// TIA Portal V20 export
DATA_BLOCK "instGetIdentRf"   // DB217
// stored: InstanceOfName GetIdentRf, InstanceOfType FB
"GetIdentRf"
   // VAR_INPUT
   //    identRfAllUnits { ExternalAccessible := 'False'; ExternalVisible := 'False'; ExternalWritable := 'False'} : Array[0.."NO_OF_UNITS"] of "typeEMIdentRf";
   //    numberOfRfReaders : USInt := 1;
   // END_VAR
   // VAR_OUTPUT
   //    selectedUnit : USInt := 1;
   //    selectedEM : USInt := 6;
   //    error : Word := 16#7001;
   // END_VAR
   // VAR_IN_OUT
   //    IdentRfInterfaceHmi : "typeIdentRfHmi";
   // END_VAR
   // VAR
   //    statSelectedEMIdentRf : USInt := 6;
   //    statSelectedUnitIdentRf : USInt := 1;
   // END_VAR
BEGIN
   identRfAllUnits[0].identRfEM[0..7].selectedUnit := 0;
   identRfAllUnits[0].identRfEM[0..7].selectedEM := 0;
   identRfAllUnits[0].identRfEM[0..7].rfReaderId := 0;
   identRfAllUnits[0].identRfEM[0..7].numberOfRf := 0;
   identRfAllUnits[0].identRfEM[0].rfReader[0..1].deviceName := WSTRING#'';
   identRfAllUnits[0].identRfEM[1].rfReader[0..1].deviceName := WSTRING#'';
   identRfAllUnits[0].identRfEM[2].rfReader[0..1].deviceName := WSTRING#'';
   identRfAllUnits[0].identRfEM[3].rfReader[0..1].deviceName := WSTRING#'';
   identRfAllUnits[0].identRfEM[4].rfReader[0..1].deviceName := WSTRING#'';
   identRfAllUnits[0].identRfEM[5].rfReader[0..1].deviceName := WSTRING#'';
   identRfAllUnits[0].identRfEM[6].rfReader[0..1].deviceName := WSTRING#'';
   identRfAllUnits[0].identRfEM[7].rfReader[0..1].deviceName := WSTRING#'';
   identRfAllUnits[0].identRfEM[0].rfReader[0..1].deviceType := WSTRING#'';
   identRfAllUnits[0].identRfEM[1].rfReader[0..1].deviceType := WSTRING#'';
   identRfAllUnits[0].identRfEM[2].rfReader[0..1].deviceType := WSTRING#'';
   identRfAllUnits[0].identRfEM[3].rfReader[0..1].deviceType := WSTRING#'';
   identRfAllUnits[0].identRfEM[4].rfReader[0..1].deviceType := WSTRING#'';
   identRfAllUnits[0].identRfEM[5].rfReader[0..1].deviceType := WSTRING#'';
   identRfAllUnits[0].identRfEM[6].rfReader[0..1].deviceType := WSTRING#'';
   identRfAllUnits[0].identRfEM[7].rfReader[0..1].deviceType := WSTRING#'';
   identRfAllUnits[0].identRfEM[0].rfReader[0..1].deviceId := 0;
   identRfAllUnits[0].identRfEM[1].rfReader[0..1].deviceId := 0;
   identRfAllUnits[0].identRfEM[2].rfReader[0..1].deviceId := 0;
   identRfAllUnits[0].identRfEM[3].rfReader[0..1].deviceId := 0;
   identRfAllUnits[0].identRfEM[4].rfReader[0..1].deviceId := 0;
   identRfAllUnits[0].identRfEM[5].rfReader[0..1].deviceId := 0;
   identRfAllUnits[0].identRfEM[6].rfReader[0..1].deviceId := 0;
   identRfAllUnits[0].identRfEM[7].rfReader[0..1].deviceId := 0;
   identRfAllUnits[0].identRfEM[0].rfReader[0..1].tagType := WSTRING#'';
   identRfAllUnits[0].identRfEM[1].rfReader[0..1].tagType := WSTRING#'';
   identRfAllUnits[0].identRfEM[2].rfReader[0..1].tagType := WSTRING#'';
   identRfAllUnits[0].identRfEM[3].rfReader[0..1].tagType := WSTRING#'';
   identRfAllUnits[0].identRfEM[4].rfReader[0..1].tagType := WSTRING#'';
   identRfAllUnits[0].identRfEM[5].rfReader[0..1].tagType := WSTRING#'';
   identRfAllUnits[0].identRfEM[6].rfReader[0..1].tagType := WSTRING#'';
   identRfAllUnits[0].identRfEM[7].rfReader[0..1].tagType := WSTRING#'';
   identRfAllUnits[0].identRfEM[0].rfReader[0..1].cameraMode := WSTRING#'';
   identRfAllUnits[0].identRfEM[1].rfReader[0..1].cameraMode := WSTRING#'';
   identRfAllUnits[0].identRfEM[2].rfReader[0..1].cameraMode := WSTRING#'';
   identRfAllUnits[0].identRfEM[3].rfReader[0..1].cameraMode := WSTRING#'';
   identRfAllUnits[0].identRfEM[4].rfReader[0..1].cameraMode := WSTRING#'';
   identRfAllUnits[0].identRfEM[5].rfReader[0..1].cameraMode := WSTRING#'';
   identRfAllUnits[0].identRfEM[6].rfReader[0..1].cameraMode := WSTRING#'';
   identRfAllUnits[0].identRfEM[7].rfReader[0..1].cameraMode := WSTRING#'';
   identRfAllUnits[0].identRfEM[0].rfReader[0..1].resultState := WSTRING#'';
   identRfAllUnits[0].identRfEM[1].rfReader[0..1].resultState := WSTRING#'';
   identRfAllUnits[0].identRfEM[2].rfReader[0..1].resultState := WSTRING#'';
   identRfAllUnits[0].identRfEM[3].rfReader[0..1].resultState := WSTRING#'';
   identRfAllUnits[0].identRfEM[4].rfReader[0..1].resultState := WSTRING#'';
   identRfAllUnits[0].identRfEM[5].rfReader[0..1].resultState := WSTRING#'';
   identRfAllUnits[0].identRfEM[6].rfReader[0..1].resultState := WSTRING#'';
   identRfAllUnits[0].identRfEM[7].rfReader[0..1].resultState := WSTRING#'';
   identRfAllUnits[0].identRfEM[0].rfReader[0..1].progNo := 0;
   identRfAllUnits[0].identRfEM[1].rfReader[0..1].progNo := 0;
   identRfAllUnits[0].identRfEM[2].rfReader[0..1].progNo := 0;
   identRfAllUnits[0].identRfEM[3].rfReader[0..1].progNo := 0;
   identRfAllUnits[0].identRfEM[4].rfReader[0..1].progNo := 0;
   identRfAllUnits[0].identRfEM[5].rfReader[0..1].progNo := 0;
   identRfAllUnits[0].identRfEM[6].rfReader[0..1].progNo := 0;
   identRfAllUnits[0].identRfEM[7].rfReader[0..1].progNo := 0;
   identRfAllUnits[0].identRfEM[0].rfReader[0..1].progNumberWrite := 0;
   identRfAllUnits[0].identRfEM[1].rfReader[0..1].progNumberWrite := 0;
   identRfAllUnits[0].identRfEM[2].rfReader[0..1].progNumberWrite := 0;
   identRfAllUnits[0].identRfEM[3].rfReader[0..1].progNumberWrite := 0;
   identRfAllUnits[0].identRfEM[4].rfReader[0..1].progNumberWrite := 0;
   identRfAllUnits[0].identRfEM[5].rfReader[0..1].progNumberWrite := 0;
   identRfAllUnits[0].identRfEM[6].rfReader[0..1].progNumberWrite := 0;
   identRfAllUnits[0].identRfEM[7].rfReader[0..1].progNumberWrite := 0;
   identRfAllUnits[0].identRfEM[0].rfReader[0..1].pushbutton := 16#0000;
   identRfAllUnits[0].identRfEM[1].rfReader[0..1].pushbutton := 16#0000;
   identRfAllUnits[0].identRfEM[2].rfReader[0..1].pushbutton := 16#0000;
   identRfAllUnits[0].identRfEM[3].rfReader[0..1].pushbutton := 16#0000;
   identRfAllUnits[0].identRfEM[4].rfReader[0..1].pushbutton := 16#0000;
   identRfAllUnits[0].identRfEM[5].rfReader[0..1].pushbutton := 16#0000;
   identRfAllUnits[0].identRfEM[6].rfReader[0..1].pushbutton := 16#0000;
   identRfAllUnits[0].identRfEM[7].rfReader[0..1].pushbutton := 16#0000;
   identRfAllUnits[0].identRfEM[0].rfReader[0..1].enablePushbutton := 16#0000;
   identRfAllUnits[0].identRfEM[1].rfReader[0..1].enablePushbutton := 16#0000;
   identRfAllUnits[0].identRfEM[2].rfReader[0..1].enablePushbutton := 16#0000;
   identRfAllUnits[0].identRfEM[3].rfReader[0..1].enablePushbutton := 16#0000;
   identRfAllUnits[0].identRfEM[4].rfReader[0..1].enablePushbutton := 16#0000;
   identRfAllUnits[0].identRfEM[5].rfReader[0..1].enablePushbutton := 16#0000;
   identRfAllUnits[0].identRfEM[6].rfReader[0..1].enablePushbutton := 16#0000;
   identRfAllUnits[0].identRfEM[7].rfReader[0..1].enablePushbutton := 16#0000;
   identRfAllUnits[0].identRfEM[0].rfReader[0..1].status := 16#0000;
   identRfAllUnits[0].identRfEM[1].rfReader[0..1].status := 16#0000;
   identRfAllUnits[0].identRfEM[2].rfReader[0..1].status := 16#0000;
   identRfAllUnits[0].identRfEM[3].rfReader[0..1].status := 16#0000;
   identRfAllUnits[0].identRfEM[4].rfReader[0..1].status := 16#0000;
   identRfAllUnits[0].identRfEM[5].rfReader[0..1].status := 16#0000;
   identRfAllUnits[0].identRfEM[6].rfReader[0..1].status := 16#0000;
   identRfAllUnits[0].identRfEM[7].rfReader[0..1].status := 16#0000;
   identRfAllUnits[0].identRfEM[0].rfReader[0..1].alarmCategorie := 0;
   identRfAllUnits[0].identRfEM[1].rfReader[0..1].alarmCategorie := 0;
   identRfAllUnits[0].identRfEM[2].rfReader[0..1].alarmCategorie := 0;
   identRfAllUnits[0].identRfEM[3].rfReader[0..1].alarmCategorie := 0;
   identRfAllUnits[0].identRfEM[4].rfReader[0..1].alarmCategorie := 0;
   identRfAllUnits[0].identRfEM[5].rfReader[0..1].alarmCategorie := 0;
   identRfAllUnits[0].identRfEM[6].rfReader[0..1].alarmCategorie := 0;
   identRfAllUnits[0].identRfEM[7].rfReader[0..1].alarmCategorie := 0;
   identRfAllUnits[0].identRfEM[0].rfReader[0..1].alarmNo := 0;
   identRfAllUnits[0].identRfEM[1].rfReader[0..1].alarmNo := 0;
   identRfAllUnits[0].identRfEM[2].rfReader[0..1].alarmNo := 0;
   identRfAllUnits[0].identRfEM[3].rfReader[0..1].alarmNo := 0;
   identRfAllUnits[0].identRfEM[4].rfReader[0..1].alarmNo := 0;
   identRfAllUnits[0].identRfEM[5].rfReader[0..1].alarmNo := 0;
   identRfAllUnits[0].identRfEM[6].rfReader[0..1].alarmNo := 0;
   identRfAllUnits[0].identRfEM[7].rfReader[0..1].alarmNo := 0;
   identRfAllUnits[0].identRfEM[0].rfReader[0..1].alarmCode := 16#0000_0000;
   identRfAllUnits[0].identRfEM[1].rfReader[0..1].alarmCode := 16#0000_0000;
   identRfAllUnits[0].identRfEM[2].rfReader[0..1].alarmCode := 16#0000_0000;
   identRfAllUnits[0].identRfEM[3].rfReader[0..1].alarmCode := 16#0000_0000;
   identRfAllUnits[0].identRfEM[4].rfReader[0..1].alarmCode := 16#0000_0000;
   identRfAllUnits[0].identRfEM[5].rfReader[0..1].alarmCode := 16#0000_0000;
   identRfAllUnits[0].identRfEM[6].rfReader[0..1].alarmCode := 16#0000_0000;
   identRfAllUnits[0].identRfEM[7].rfReader[0..1].alarmCode := 16#0000_0000;
   identRfAllUnits[0].identRfEM[0].rfReader[0..1].resultColor := 0;
   identRfAllUnits[0].identRfEM[1].rfReader[0..1].resultColor := 0;
   identRfAllUnits[0].identRfEM[2].rfReader[0..1].resultColor := 0;
   identRfAllUnits[0].identRfEM[3].rfReader[0..1].resultColor := 0;
   identRfAllUnits[0].identRfEM[4].rfReader[0..1].resultColor := 0;
   identRfAllUnits[0].identRfEM[5].rfReader[0..1].resultColor := 0;
   identRfAllUnits[0].identRfEM[6].rfReader[0..1].resultColor := 0;
   identRfAllUnits[0].identRfEM[7].rfReader[0..1].resultColor := 0;
   identRfAllUnits[0].identRfEM[0].rfReader[0..1].statusColorCode := 0;
   identRfAllUnits[0].identRfEM[1].rfReader[0..1].statusColorCode := 0;
   identRfAllUnits[0].identRfEM[2].rfReader[0..1].statusColorCode := 0;
   identRfAllUnits[0].identRfEM[3].rfReader[0..1].statusColorCode := 0;
   identRfAllUnits[0].identRfEM[4].rfReader[0..1].statusColorCode := 0;
   identRfAllUnits[0].identRfEM[5].rfReader[0..1].statusColorCode := 0;
   identRfAllUnits[0].identRfEM[6].rfReader[0..1].statusColorCode := 0;
   identRfAllUnits[0].identRfEM[7].rfReader[0..1].statusColorCode := 0;
   identRfAllUnits[0].identRfEM[0].rfReader[0..1].datRead1 := '';
   identRfAllUnits[0].identRfEM[1].rfReader[0..1].datRead1 := '';
   identRfAllUnits[0].identRfEM[2].rfReader[0..1].datRead1 := '';
   identRfAllUnits[0].identRfEM[3].rfReader[0..1].datRead1 := '';
   identRfAllUnits[0].identRfEM[4].rfReader[0..1].datRead1 := '';
   identRfAllUnits[0].identRfEM[5].rfReader[0..1].datRead1 := '';
   identRfAllUnits[0].identRfEM[6].rfReader[0..1].datRead1 := '';
   identRfAllUnits[0].identRfEM[7].rfReader[0..1].datRead1 := '';
   identRfAllUnits[0].identRfEM[0].rfReader[0..1].datRead2 := '';
   identRfAllUnits[0].identRfEM[1].rfReader[0..1].datRead2 := '';
   identRfAllUnits[0].identRfEM[2].rfReader[0..1].datRead2 := '';
   identRfAllUnits[0].identRfEM[3].rfReader[0..1].datRead2 := '';
   identRfAllUnits[0].identRfEM[4].rfReader[0..1].datRead2 := '';
   identRfAllUnits[0].identRfEM[5].rfReader[0..1].datRead2 := '';
   identRfAllUnits[0].identRfEM[6].rfReader[0..1].datRead2 := '';
   identRfAllUnits[0].identRfEM[7].rfReader[0..1].datRead2 := '';
   identRfAllUnits[0].identRfEM[0].rfReader[0..1].datRead3 := '';
   identRfAllUnits[0].identRfEM[1].rfReader[0..1].datRead3 := '';
   identRfAllUnits[0].identRfEM[2].rfReader[0..1].datRead3 := '';
   identRfAllUnits[0].identRfEM[3].rfReader[0..1].datRead3 := '';
   identRfAllUnits[0].identRfEM[4].rfReader[0..1].datRead3 := '';
   identRfAllUnits[0].identRfEM[5].rfReader[0..1].datRead3 := '';
   identRfAllUnits[0].identRfEM[6].rfReader[0..1].datRead3 := '';
   identRfAllUnits[0].identRfEM[7].rfReader[0..1].datRead3 := '';
   identRfAllUnits[0].identRfEM[0].rfReader[0..1].datRead4 := '';
   identRfAllUnits[0].identRfEM[1].rfReader[0..1].datRead4 := '';
   identRfAllUnits[0].identRfEM[2].rfReader[0..1].datRead4 := '';
   identRfAllUnits[0].identRfEM[3].rfReader[0..1].datRead4 := '';
   identRfAllUnits[0].identRfEM[4].rfReader[0..1].datRead4 := '';
   identRfAllUnits[0].identRfEM[5].rfReader[0..1].datRead4 := '';
   identRfAllUnits[0].identRfEM[6].rfReader[0..1].datRead4 := '';
   identRfAllUnits[0].identRfEM[7].rfReader[0..1].datRead4 := '';
   identRfAllUnits[0].identRfEM[0].rfReader[0..1].datWrite1 := '';
   identRfAllUnits[0].identRfEM[1].rfReader[0..1].datWrite1 := '';
   identRfAllUnits[0].identRfEM[2].rfReader[0..1].datWrite1 := '';
   identRfAllUnits[0].identRfEM[3].rfReader[0..1].datWrite1 := '';
   identRfAllUnits[0].identRfEM[4].rfReader[0..1].datWrite1 := '';
   identRfAllUnits[0].identRfEM[5].rfReader[0..1].datWrite1 := '';
   identRfAllUnits[0].identRfEM[6].rfReader[0..1].datWrite1 := '';
   identRfAllUnits[0].identRfEM[7].rfReader[0..1].datWrite1 := '';
   identRfAllUnits[0].identRfEM[0].rfReader[0..1].datWrite2 := '';
   identRfAllUnits[0].identRfEM[1].rfReader[0..1].datWrite2 := '';
   identRfAllUnits[0].identRfEM[2].rfReader[0..1].datWrite2 := '';
   identRfAllUnits[0].identRfEM[3].rfReader[0..1].datWrite2 := '';
   identRfAllUnits[0].identRfEM[4].rfReader[0..1].datWrite2 := '';
   identRfAllUnits[0].identRfEM[5].rfReader[0..1].datWrite2 := '';
   identRfAllUnits[0].identRfEM[6].rfReader[0..1].datWrite2 := '';
   identRfAllUnits[0].identRfEM[7].rfReader[0..1].datWrite2 := '';
   identRfAllUnits[0].identRfEM[0].rfReader[0..1].datWrite3 := '';
   identRfAllUnits[0].identRfEM[1].rfReader[0..1].datWrite3 := '';
   identRfAllUnits[0].identRfEM[2].rfReader[0..1].datWrite3 := '';
   identRfAllUnits[0].identRfEM[3].rfReader[0..1].datWrite3 := '';
   identRfAllUnits[0].identRfEM[4].rfReader[0..1].datWrite3 := '';
   identRfAllUnits[0].identRfEM[5].rfReader[0..1].datWrite3 := '';
   identRfAllUnits[0].identRfEM[6].rfReader[0..1].datWrite3 := '';
   identRfAllUnits[0].identRfEM[7].rfReader[0..1].datWrite3 := '';
   identRfAllUnits[0].identRfEM[0].rfReader[0..1].datWrite4 := '';
   identRfAllUnits[0].identRfEM[1].rfReader[0..1].datWrite4 := '';
   identRfAllUnits[0].identRfEM[2].rfReader[0..1].datWrite4 := '';
   identRfAllUnits[0].identRfEM[3].rfReader[0..1].datWrite4 := '';
   identRfAllUnits[0].identRfEM[4].rfReader[0..1].datWrite4 := '';
   identRfAllUnits[0].identRfEM[5].rfReader[0..1].datWrite4 := '';
   identRfAllUnits[0].identRfEM[6].rfReader[0..1].datWrite4 := '';
   identRfAllUnits[0].identRfEM[7].rfReader[0..1].datWrite4 := '';
END_DATA_BLOCK
